FUNCTION_BLOCK FB_WriteParameterNC_TestDouble IMPLEMENTS  I_WriteParameter
VAR_INPUT
END_VAR
VAR_OUTPUT
END_VAR
VAR
END_VAR

{warning 'Add property implementation'}
PROPERTY Aborted : BOOL
GET
END_GET
END_PROPERTY

{warning 'Add property implementation'}
PROPERTY Active : BOOL
GET
END_GET
END_PROPERTY

{warning 'Add property implementation'}
PROPERTY Busy : BOOL
GET
END_GET
END_PROPERTY

{warning 'Add property implementation'}
PROPERTY Done : BOOL
GET
END_GET
END_PROPERTY

{warning 'Add property implementation'}
PROPERTY Error : BOOL
GET
END_GET
END_PROPERTY

{warning 'Add property implementation'}
PROPERTY ErrorID : UDINT
GET
END_GET
END_PROPERTY

{warning 'Add property implementation'}
PROPERTY Message : T_MAXSTRING
GET
END_GET
END_PROPERTY

{warning 'Add method implementation '}
METHOD WriteParameter
VAR_INPUT
    Execute	: BOOL;
    ParameterNumber	: MC_AxisParameter;
    ParameterValue	: LREAL;
END_VAR
END_METHOD

END_FUNCTION_BLOCK

(* stored: Version 1.1.0.1
   POU FB_WriteParameterNC_TestDouble: Id {585873b6-7f78-428d-a151-a1ef70c92da6}, SpecialFunc None
   Property Aborted: Id {7396920b-2600-424f-9c6c-770311b58147}
   Get Get: Id {c8e136ef-2c49-45f2-835f-402f6de965d7}
   Property Active: Id {a386a0b0-2594-44cc-8652-b40c3432108f}
   Get Get: Id {2a23fc67-b513-4551-9c11-33d28ec4831e}
   Property Busy: Id {ee2addf4-3000-45bf-93ee-5c6d9199c1f3}
   Get Get: Id {d7030bbf-37ba-4166-8a3b-c535d58f2b7f}
   Property Done: Id {285e3e5d-9d50-4f87-ac74-f6629d45e656}
   Get Get: Id {4f5689bb-076c-40a7-bd20-ace516750671}
   Property Error: Id {062ba1c5-be7a-4fe9-8b23-dcf7b5a13d3a}
   Get Get: Id {24f0f280-919f-4cac-bd35-881b4630d462}
   Property ErrorID: Id {874f763c-3159-412b-99e6-d6549eeb89d8}
   Get Get: Id {89605898-8cb2-4fb2-b49e-b1d0641a8bee}
   Property Message: Id {98221eac-3ece-43a4-8c71-2195803f72fb}
   Get Get: Id {63537d90-ad5e-4a72-89fb-9e94f99a34f5}
   Method WriteParameter: Id {7d0bfa80-d3f9-4353-95de-f3619b083423} *)
